// TIA Portal V16 export
// export: Created 2021-11-15T20:32:30.2361424Z, ExportSetting WithDefaults, DisplayName Totally Integrated Automation Portal, DisplayVersion V16, DisplayName TIA Portal Version Control Interface, DisplayVersion V16, DisplayName TIA Portal Openness, DisplayVersion V16, DisplayName TIA Portal Teamcenter Gateway, DisplayVersion V16, DisplayName STEP 7 Professional, DisplayVersion V16, DisplayName STEP 7 Safety, DisplayVersion V16, DisplayName WinCC Professional, DisplayVersion V16
VAR_GLOBAL   // PLC tag table "Table de variables standard"
   Bascule AT %M0.0 : Bool;
   Bit1 AT %M0.1 : Bool;
   Bit2 AT %M0.2 : Bool;
   Bit3 AT %M0.3 : Bool;
   Sensor1 AT %M0.4 : Bool;
   Sensor2 AT %M0.5 : Bool;
   Coil20 AT %M0.6 : Bool;
END_VAR
